// SIMATIC S7-200 project (STEP 7-Micro/WIN), CPU 226 REL 01.23

ORGANIZATION_BLOCK MAIN:OB1
TITLE=The system initiates the mixing process through a start button, opening feed valve A and feed valve B respectively to begin feeding. Feed valve A operates only when level sensor A does not detect a full level and the safety sensor does not trigger an alarm; similarly, feed valve B operates only when level sensor B does not detect a full level and the safety sensor remains unalarmed. During the feeding process, temperature sensor A activates the heater control via a signal, while temperature sensor B activates the cooler control via a signal. Once feeding is complete, mixing motor A and mixing motor B start separately, with their operation durations controlled by mixing timer A and mixing timer B, respectively, set to 100 time units. After mixing concludes, the control signal for discharge valve A triggers it to open, and the control signal for discharge valve B triggers it to open, with the discharge times managed by discharge timer A and discharge timer B, respectively, set to 5 time units each. A manual mode switch and an automatic mode switch allow the operator to choose the preferred operation mode. The system records the discharge status using status flag A and status flag B.
BEGIN
Network 1 // Network Title
// Network Comment
LD     I10.5
CALL   SBR_7:SBR7
Network 2
LD     I10.2
CALL   SBR_8:SBR8
Network 3
LD     I10.3
CALL   SBR_0:SBR0
Network 4
LD     I10.0
CALL   SBR_2:SBR2
Network 5
LD     I10.4
O      I10.1
CALL   SBR_4:SBR4
Network 6
LD     SM0.0
CALL   SBR_6:SBR6
Network 7
LD     I10.2
O      I10.5
=      L60.0
LD     M23.0
AN     I1.6
LD     M23.1
AN     I1.0
OLD
LD     M23.1
AN     I1.1
OLD
LD     M23.1
AN     I1.1
OLD
=      L63.7
LD     L60.0
CALL   SBR_9:SBR9, L63.7, Q3.3, Q3.0, Q3.4, Q3.1
Network 8
LD     SM0.0
CALL   SBR_5:SBR5
Network 9
LD     I10.3
O      I10.0
CALL   SBR_10:SBR10
END_ORGANIZATION_BLOCK

SUBROUTINE_BLOCK SBR_0:SBR0
TITLE=POU Comment
BEGIN
Network 1 // Network Title
// Network Comment
LD     I8.6
AN     I3.5
A      I1.6
AN     Q2.7
=      Q2.3
Network 2
LD     I11.4
EU
O      Q1.3
AN     I1.6
AN     Q1.6
AN     I7.2
AN     T46
=      Q1.3
Network 3
LD     Q1.3
TON    T46, +100
Network 4
LD     Q1.3
ED
O      Q6.6
AN     Q1.6
=      Q6.6
Network 5
LD     I11.5
EU
O      Q1.6
A      I1.6
AN     Q1.3
AN     I7.2
AN     T47
=      Q1.6
Network 6
LD     Q1.6
TON    T47, +100
Network 7
LD     Q1.6
ED
O      Q6.7
AN     Q1.3
=      Q6.7
Network 9
LD     I8.7
AN     I3.5
A      I1.7
AN     Q2.3
AN     Q3.1
AN     Q3.0
=      Q2.7
END_SUBROUTINE_BLOCK

SUBROUTINE_BLOCK SBR_1:SBR1
TITLE=
VAR_INPUT
ZMTT_xj:BOOL;	// L0.0 
ZMTT_xx:BOOL;	// L0.1 
ZMTT_ss:BOOL;	// L0.2 
ZMTT_sx:BOOL;	// L0.3 
END_VAR
VAR_OUTPUT
ZMTT_s:BOOL;	// L0.4 
ZMTT_x:BOOL;	// L0.5 
END_VAR
BEGIN
Network 1
LD     #ZMTT_xj:L0.0
AN     I3.5
A      #ZMTT_xx:L0.1
AN     #ZMTT_s:L0.4
=      #ZMTT_x:L0.5
Network 2
LD     #ZMTT_ss:L0.2
AN     I3.5
A      #ZMTT_sx:L0.3
AN     #ZMTT_x:L0.5
=      #ZMTT_s:L0.4
END_SUBROUTINE_BLOCK

SUBROUTINE_BLOCK SBR_2:SBR2
TITLE=
BEGIN
Network 1
LD     SM0.0
=      L60.0
LD     I8.0
=      L63.7
LD     I1.0
=      L63.6
LD     I8.3
=      L63.5
LD     I1.3
=      L63.4
LD     L60.0
CALL   SBR_1:SBR1, L63.7, L63.6, L63.5, L63.4, Q2.4, Q2.0
Network 2
LD     SM0.0
=      L60.0
LD     I8.1
=      L63.7
LD     I1.1
=      L63.6
LD     I8.4
=      L63.5
LD     I1.4
=      L63.4
LD     L60.0
CALL   SBR_1:SBR1, L63.7, L63.6, L63.5, L63.4, Q2.5, Q2.1
Network 3
LD     SM0.0
=      L60.0
LD     I8.2
=      L63.7
LD     I1.2
=      L63.6
LD     I8.5
=      L63.5
LD     I1.5
=      L63.4
LD     L60.0
CALL   SBR_1:SBR1, L63.7, L63.6, L63.5, L63.4, Q2.6, Q2.2
Network 4
LD     SM0.0
CALL   SBR_3:SBR3
END_SUBROUTINE_BLOCK

SUBROUTINE_BLOCK SBR_3:SBR3
TITLE=
BEGIN
Network 1
LD     I11.0
EU
O      Q1.1
AN     I0.0
AN     I7.0
AN     Q1.4
AN     I1.0
AN     I1.1
AN     I3.5
=      Q1.1
Network 2
LD     I11.1
EU
O      Q1.4
AN     I0.1
AN     I7.0
AN     Q1.1
=      Q1.4
Network 3
LD     I11.2
EU
O      Q1.2
AN     I0.4
AN     I7.1
AN     Q1.5
AN     I1.0
AN     I1.1
AN     I3.5
=      Q1.2
Network 4
LD     I11.3
EU
O      Q1.5
AN     I0.5
AN     I7.1
AN     Q1.2
=      Q1.5
END_SUBROUTINE_BLOCK

SUBROUTINE_BLOCK SBR_4:SBR4
TITLE=
BEGIN
Network 1
LD     I8.6
A      I1.6
AN     Q2.7
=      Q2.3
Network 2
LD     I8.7
A      I1.7
AN     Q2.3
=      Q2.7
Network 3
LD     I11.4
O      Q1.3
AN     I7.2
AN     Q1.6
AN     T48
=      Q1.3
Network 4
LD     Q1.3
TON    T48, +100
Network 5
LD     Q1.3
ED
O      Q5.6
AN     Q1.6
=      Q5.6
Network 6
LD     Q1.6
ED
O      Q5.7
AN     Q1.3
=      Q5.7
Network 7
LD     I11.5
O      Q1.6
AN     I7.2
AN     Q1.3
AN     T49
=      Q1.6
Network 8
LD     Q1.6
TON    T49, +100
Network 9
LD     I8.0
A      I1.0
AN     Q2.4
=      Q2.0
Network 10
LD     I8.3
A      I1.3
AN     Q2.0
=      Q2.4
Network 11
LD     I11.0
O      Q1.1
AN     I7.0
AN     I0.0
AN     Q1.4
=      Q1.1
Network 12
LD     I11.2
O      Q1.2
AN     I7.1
AN     I0.4
AN     Q1.5
=      Q1.2
Network 13
LD     I11.1
O      Q1.4
AN     I7.0
AN     I0.1
AN     Q1.1
=      Q1.4
Network 14
LD     I11.3
O      Q1.5
AN     I7.1
AN     I0.5
AN     Q1.2
=      Q1.5
Network 15
LD     I8.1
A      I1.1
AN     Q2.5
=      Q2.1
Network 16
LD     I8.4
A      I1.4
AN     Q2.1
=      Q2.5
Network 17
LD     I8.2
A      I1.2
AN     Q2.6
=      Q2.2
Network 18
LD     I8.5
A      I1.5
AN     Q2.2
=      Q2.6
Network 20
LD     I9.0
O      M4.1
AN     Q3.3
A      I2.6
AN     Q3.0
=      M4.1
TON    T58, +5
Network 21
LD     T58
O      Q3.3
AN     I7.5
AN     Q3.0
A      I2.6
AN     I9.1
=      Q3.3
S      M4.2, 1
Network 22
LD     I9.1
O      M4.0
AN     Q3.3
AN     Q3.0
A      I2.6
A      I1.0
LPS
A      M4.2
=      M4.0
LPP
TON    T59, +5
Network 23
LD     T59
O      Q3.0
AN     I7.5
AN     Q3.3
A      I2.6
AN     I9.0
=      Q3.0
Network 24
LD     I7.5
R      M4.2, 1
Network 25
LD     I9.2
O      M4.5
AN     Q3.4
A      I2.7
AN     Q3.1
=      M4.5
TON    T60, +5
Network 26
LD     T60
O      Q3.4
AN     I7.6
AN     Q3.1
A      I2.7
AN     I9.3
=      Q3.4
S      M4.6, 1
Network 27
LD     I9.3
O      M4.4
AN     Q3.4
AN     Q3.1
A      I2.7
A      I1.0
LPS
A      M4.6
=      M4.4
LPP
TON    T61, +5
Network 28
LD     T61
O      Q3.1
AN     I7.6
AN     Q3.4
A      I2.7
AN     I9.2
=      Q3.1
Network 29
LD     I7.6
R      M4.6, 1
END_SUBROUTINE_BLOCK

SUBROUTINE_BLOCK SBR_5:SBR5
TITLE=
BEGIN
Network 1
LD     I9.6
O      Q0.0
AN     I7.3
AN     I3.5
=      Q0.0
Network 2
LD     I9.7
O      Q0.1
AN     I7.4
AN     I3.5
=      Q0.1
Network 3
LD     I6.7
O      Q3.2
AN     I10.7
A      Q0.0
=      Q3.2
Network 4
LD     I6.6
O      Q3.5
AN     I7.7
A      Q0.1
=      Q3.5
END_SUBROUTINE_BLOCK

SUBROUTINE_BLOCK SBR_6:SBR6
TITLE=
BEGIN
Network 1
LD     I10.6
O      I3.2
=      Q4.3
Network 2
LD     I10.6
O      I2.4
=      Q4.5
Network 3
LD     I10.6
O      I2.5
=      Q4.6
Network 4
LD     I10.6
O      I3.3
=      Q4.7
Network 5
LD     I10.6
O      I3.0
=      Q5.0
Network 6
LD     I10.6
O      I3.1
=      Q5.1
Network 7
LD     I10.6
O      I2.1
=      Q5.2
Network 8
LD     I10.6
O      I2.2
=      Q5.3
Network 9
LD     I10.6
ON     I0.1
=      Q6.0
Network 10
LD     I10.6
ON     I0.5
=      Q6.1
Network 11
LD     I10.6
LD     I10.3
A      Q6.6
OLD
LD     I10.1
A      Q5.6
OLD
O      M8.0
=      Q6.2
Network 12
LD     I10.6
ON     I0.0
=      Q6.3
Network 13
LD     I10.6
ON     I0.4
=      Q6.4
Network 14
LD     I10.6
LD     I10.3
A      Q6.7
OLD
LD     I10.1
A      Q5.7
OLD
O      M8.1
=      Q6.5
Network 15
LD     I10.6
ON     I1.0
=      Q7.0
Network 16
LD     I10.6
ON     I1.1
=      Q7.1
Network 17
LD     I10.6
ON     I1.2
=      Q7.2
Network 18
LD     I10.6
ON     I1.3
=      Q7.3
Network 19
LD     I10.6
ON     I1.4
=      Q7.4
Network 20
LD     I10.6
ON     I1.5
=      Q7.5
Network 21
LD     I10.6
ON     I1.7
=      Q7.6
Network 22
LD     I10.6
ON     I1.6
=      Q7.7
Network 23
LDN    I1.3
AN     I1.4
AN     I1.5
AN     I1.7
AN     I0.3
=      Q3.6
Network 24
LD     I10.6
O      Q3.6
=      Q0.4
Network 25
LD     I6.0
=      Q0.5
Network 26
LD     I6.1
=      Q0.6
Network 27
LD     I0.3
=      Q0.2
END_SUBROUTINE_BLOCK

SUBROUTINE_BLOCK SBR_7:SBR7
TITLE=
BEGIN
Network 1
LD     I8.6
O      Q2.3
AN     I3.5
A      I1.6
AN     Q2.7
=      Q2.3
Network 2
LD     I2.6
A      I2.7
=      M12.4
A      I3.0
TON    T120, +100
Network 3
LD     I3.0
A      I2.6
AN     M12.4
TON    T121, +100
Network 4
LD     I3.1
A      I2.7
AN     M12.4
TON    T122, +100
Network 5
LD     T120
O      T121
O      T122
EU
O      Q1.3
AN     T50
AN     Q1.6
=      Q1.3
Network 6
LD     I8.7
O      Q2.7
AN     I3.5
A      I1.7
AN     Q2.3
=      Q2.7
Network 7
LD     Q2.7
O      Q1.6
AN     T130
AN     Q1.3
=      Q1.6
Network 8
LD     Q1.6
TON    T130, +200
Network 9
LD     Q1.3
TON    T50, +200
Network 10
LD     Q1.3
ED
O      M8.0
AN     Q1.6
=      M8.0
Network 11
LD     Q1.6
ED
O      M8.1
AN     Q1.3
=      M8.1
END_SUBROUTINE_BLOCK

SUBROUTINE_BLOCK SBR_8:SBR8
TITLE=
BEGIN
Network 1
LD     I8.0
O      Q2.0
O      I8.1
O      I8.2
AN     I3.5
A      I1.0
AN     Q2.4
=      Q2.0
Network 2
LD     I3.0
AN     I2.7
O      I3.1
TON    T132, +200
Network 3
LD     T132
EU
O      Q1.1
AN     I0.0
AN     I7.0
AN     Q1.4
=      Q1.1
Network 4
LD     I8.3
O      Q2.4
O      I8.4
O      I8.4
AN     I3.5
A      I1.3
AN     Q2.0
=      Q2.4
Network 5
LD     Q2.4
EU
O      Q1.4
AN     I0.1
AN     I7.0
AN     Q1.1
=      Q1.4
Network 6
LD     I8.1
O      Q2.1
O      I8.0
O      I8.2
AN     I3.5
A      I1.1
AN     Q2.5
=      Q2.1
Network 7
LD     T132
EU
O      Q1.2
AN     I0.4
AN     I7.1
AN     Q1.5
=      Q1.2
Network 8
LD     I8.4
O      Q2.5
O      I8.3
O      I8.5
AN     I3.5
A      I1.4
AN     Q2.1
=      Q2.5
Network 9
LD     Q2.5
EU
O      Q1.5
AN     I0.5
AN     I7.1
AN     Q1.2
=      Q1.5
Network 10
LD     I8.2
O      Q2.2
O      I8.1
O      I8.0
AN     I3.5
A      I1.2
AN     Q2.6
=      Q2.2
Network 11
LD     I8.5
O      Q2.6
O      I8.4
O      I8.3
AN     I3.5
A      I1.5
AN     Q2.2
=      Q2.6
END_SUBROUTINE_BLOCK

SUBROUTINE_BLOCK SBR_9:SBR9
TITLE=
VAR_INPUT
KS_GS:BOOL;	// L0.0 
END_VAR
VAR_OUTPUT
FJ1_DS:BOOL;	// L0.1 
FJ1_GS:BOOL;	// L0.2 
FJ2_DS:BOOL;	// L0.3 
FJ2_GS:BOOL;	// L0.4 
END_VAR
BEGIN
Network 1
LD     I9.0
O      #FJ1_DS:L0.1
O      T55
LPS
AN     I7.5
A      M20.4
A      I2.6
AN     #KS_GS:L0.0
=      #FJ1_DS:L0.1
LPP
S      M20.4, 1
Network 2
LD     I8.6
S      M23.0, 1
Network 3
LD     I8.7
R      M23.0, 1
Network 4
LD     I8.0
O      I8.1
O      I8.2
S      M23.1, 1
Network 5
LD     I8.3
O      I8.4
O      I8.5
R      M23.1, 1
Network 6
LD     #KS_GS:L0.0
TON    T131, +400
Network 7
LD     I9.2
O      #FJ2_DS:L0.3
O      T57
LPS
A      M20.5
AN     I7.6
A      I2.7
AN     T131
=      #FJ2_DS:L0.3
LPP
S      M20.5, 1
Network 8
LD     #KS_GS:L0.0
LPS
A      M20.4
A      I2.6
TON    T54, +5
LPP
A      M20.5
A      I2.7
TON    T56, +405
Network 9
LD     T54
A      M20.4
=      #FJ1_GS:L0.2
Network 10
LD     #KS_GS:L0.0
ED
LD     M20.2
AN     SM0.1
OLD
AN     #FJ1_DS:L0.1
LPS
A      M20.4
=      M20.2
LPP
A      I2.6
TON    T55, +10
Network 11
LD     T56
A      M20.5
=      #FJ2_GS:L0.4
Network 12
LD     #KS_GS:L0.0
ED
LD     M20.3
AN     SM0.1
OLD
AN     #FJ2_DS:L0.3
LPS
A      M20.5
=      M20.3
LPP
A      I2.7
TON    T57, +10
Network 13
LD     I7.5
R      M20.4, 1
Network 14
LD     I7.6
R      M20.5, 1
END_SUBROUTINE_BLOCK

SUBROUTINE_BLOCK SBR_10:SBR10
TITLE=
BEGIN
Network 1
LD     I9.0
O      M0.1
AN     T38
A      I2.6
AN     Q3.0
=      M0.1
TON    T38, +5
Network 2
LD     T38
O      Q3.3
AN     I7.5
AN     Q3.0
A      I2.6
AN     I9.1
=      Q3.3
S      M0.2, 1
Network 3
LD     I9.1
O      M0.0
AN     Q3.3
A      I2.6
AN     Q3.0
LPS
A      M0.2
=      M0.0
LPP
TON    T37, +5
Network 4
LD     T37
O      Q3.0
AN     I7.5
AN     Q3.3
A      I2.6
AN     I9.0
=      Q3.0
Network 5
LD     I7.5
R      M0.2, 1
Network 6
LD     I9.2
O      M0.5
AN     Q3.4
A      I2.7
AN     Q3.1
=      M0.5
TON    T39, +5
Network 7
LD     T39
O      Q3.4
AN     I7.6
AN     Q3.1
A      I2.7
AN     I9.3
=      Q3.4
S      M0.6, 1
Network 8
LD     I9.3
O      M0.4
AN     Q3.4
A      I2.7
AN     Q3.1
LPS
A      M0.6
=      M0.4
LPP
TON    T40, +5
Network 9
LD     T40
O      Q3.1
AN     I7.6
AN     Q3.4
A      I2.7
AN     I9.2
=      Q3.1
Network 10
LD     I7.6
R      M0.6, 1
END_SUBROUTINE_BLOCK
